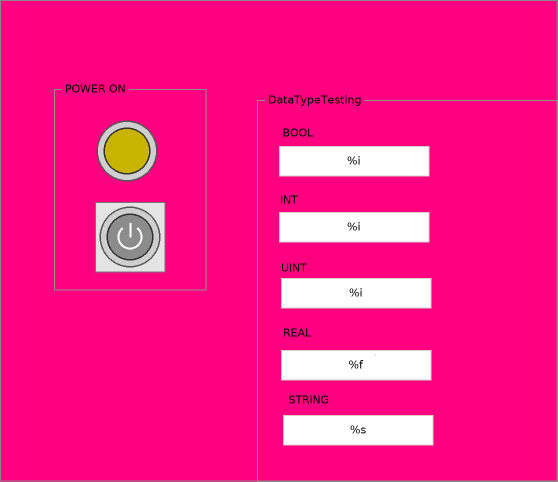
VISUALIZATION Visualization  // 558x482
    GroupBox (54,81 152x209), "POWER ON"
        Lamp1 (38,35 70x70), variable: MAIN.bEnable, style: Lamp-Lamp1-Yellow
        PowerSwitch (41,121 70x70), variable: MAIN.bStart, behaviour: TOGGLE, style: Switch-PowerSwitch-Gray
    GroupBox (257,92 301x390), "DataTypeTesting"
        Textfield (22,120 150x30), "%i", text variable: MAIN.nInt
        Textfield (22,54 150x30), "%i", text variable: MAIN.bEnable
        Textfield (24,186 150x30), "%i", text variable: MAIN.nUint
        Textfield (24,258 150x30), "%f", text variable: MAIN.fReal
            OnMouseDown: write the text variable via Edit
        Textfield (26,323 150x30), "%s", text variable: MAIN.sPowerstatus
            OnMouseDown: write the text variable via Default
            OnMouseDown: write the text variable via Default
    Label (223,118 150x30), "BOOL"
    Label (214,185 150x30), "INT"
    Label (219,253 150x30), "UINT"
    Label (222,318 150x30), "REAL"
    Label (234,385 150x30), "STRING"
    Polygon (375,355) (375,355)
END_VISUALIZATION

(* stored: Version 1.1.0.1, ProductVersion 3.1.4024.12
   Visu Visualization: Id {2d4ad43e-478f-46a7-8667-22e3ee65cbd8} *)
